  MoveL 676 to (191.54, 223.77, -20.05) mm, rotated rx -180 ry 0 rz 179.9 deg; joints [20.767, -38.825, 103.576, -157.088, 65.575, 170.653]
  MoveL 677 to (191.29, 223.93, -20.05) mm, rotated rx 180 ry 0 rz 179.9 deg; joints [20.765, -38.836, 103.603, -157.094, 65.589, 170.66]
  MoveL 678 to (191.03, 224.08, -20.05) mm, rotated rx 180 ry 0 rz 179.9 deg; joints [20.763, -38.848, 103.63, -157.098, 65.603, 170.667]
  MoveL 679 to (190.78, 224.2, -20.05) mm, rotated rx -180 ry 0 rz 179.9 deg; joints [20.762, -38.859, 103.656, -157.102, 65.617, 170.674]
  MoveL 680 to (190.53, 224.3, -20.05) mm, rotated rx 180 ry 0 rz 179.9 deg; joints [20.762, -38.87, 103.681, -157.105, 65.63, 170.681]
  MoveL 681 to (190.28, 224.39, -20.05) mm, rotated rx -180 ry 0 rz 179.9 deg; joints [20.762, -38.88, 103.706, -157.107, 65.643, 170.686]
  MoveL 682 to (190.02, 224.47, -20.05) mm, rotated rx -180 ry 0 rz 179.9 deg; joints [20.763, -38.891, 103.731, -157.109, 65.656, 170.692]
  MoveL 683 to (189.72, 224.54, -20.05) mm, rotated rx 180 ry 0 rz 179.9 deg; joints [20.765, -38.903, 103.759, -157.11, 65.672, 170.699]
  MoveL 684 to (189.41, 224.59, -20.05) mm, rotated rx -180 ry 0 rz 179.9 deg; joints [20.767, -38.915, 103.788, -157.11, 65.687, 170.704]
  MoveL 685 to (189.1, 224.63, -20.05) mm, rotated rx 180 ry 0 rz 179.9 deg; joints [20.77, -38.927, 103.815, -157.11, 65.702, 170.71]
  MoveL 686 to (188.8, 224.64, -20.05) mm, rotated rx -180 ry 0 rz 179.9 deg; joints [20.774, -38.939, 103.842, -157.108, 65.717, 170.715]
  MoveL 687 to (187.57, 224.64, -20.05) mm, rotated rx 180 ry 0 rz 179.9 deg; joints [20.79, -38.984, 103.949, -157.101, 65.775, 170.734]
  MoveL 688 to (-182.67, 224.64, -20.05) mm, rotated rx -180 ry 0 rz 179.9 deg; joints [27.375, -50.07, 132.248, -152.35, 82.128, 176.591]
  MoveL 689 to (-188.8, 224.64, -20.05) mm, rotated rx 180 ry 0 rz 179.9 deg; joints [27.516, -50.21, 132.665, -152.225, 82.383, 176.704]
  MoveL 690 to (-189.1, 224.63, -20.05) mm, rotated rx -180 ry 0 rz 179.9 deg; joints [27.524, -50.217, 132.685, -152.219, 82.395, 176.71]
  MoveL 691 to (-189.41, 224.59, -20.05) mm, rotated rx -180 ry 0 rz 179.9 deg; joints [27.532, -50.223, 132.705, -152.211, 82.407, 176.715]
  MoveL 692 to (-189.72, 224.54, -20.05) mm, rotated rx 180 ry 0 rz 179.9 deg; joints [27.542, -50.23, 132.724, -152.202, 82.419, 176.72]
  MoveL 693 to (-190.02, 224.47, -20.05) mm, rotated rx 180 ry 0 rz 179.9 deg; joints [27.552, -50.236, 132.742, -152.192, 82.43, 176.724]
  MoveL 694 to (-190.28, 224.39, -20.05) mm, rotated rx -180 ry 0 rz 179.9 deg; joints [27.561, -50.241, 132.757, -152.184, 82.439, 176.728]
  MoveL 695 to (-190.53, 224.3, -20.05) mm, rotated rx -180 ry 0 rz 179.9 deg; joints [27.571, -50.245, 132.771, -152.174, 82.448, 176.731]
  MoveL 696 to (-190.78, 224.2, -20.05) mm, rotated rx -180 ry 0 rz 179.9 deg; joints [27.582, -50.25, 132.784, -152.164, 82.457, 176.734]
  MoveL 697 to (-191.03, 224.08, -20.05) mm, rotated rx -180 ry 0 rz 179.9 deg; joints [27.593, -50.254, 132.797, -152.153, 82.465, 176.736]
  MoveL 698 to (-191.28, 223.93, -20.05) mm, rotated rx 180 ry 0 rz 179.9 deg; joints [27.605, -50.258, 132.809, -152.142, 82.473, 176.739]
  MoveL 699 to (-191.54, 223.77, -20.05) mm, rotated rx -180 ry 0 rz 179.9 deg; joints [27.618, -50.262, 132.82, -152.129, 82.48, 176.741]
  MoveL 700 to (-191.79, 223.59, -20.05) mm, rotated rx 180 ry 0 rz 179.9 deg; joints [27.632, -50.266, 132.831, -152.115, 82.487, 176.743]
  MoveL 701 to (-192.04, 223.38, -20.05) mm, rotated rx 180 ry 0 rz 179.9 deg; joints [27.647, -50.269, 132.841, -152.1, 82.493, 176.744]
  MoveL 702 to (-192.27, 223.16, -20.05) mm, rotated rx -180 ry 0 rz 179.9 deg; joints [27.662, -50.272, 132.849, -152.086, 82.499, 176.744]
  MoveL 703 to (-192.48, 222.94, -20.05) mm, rotated rx -180 ry 0 rz 179.9 deg; joints [27.677, -50.274, 132.855, -152.071, 82.503, 176.745]
  MoveL 704 to (-192.68, 222.69, -20.05) mm, rotated rx -180 ry 0 rz 179.9 deg; joints [27.693, -50.276, 132.86, -152.055, 82.507, 176.744]
  MoveL 705 to (-192.86, 222.44, -20.05) mm, rotated rx 180 ry 0 rz 179.9 deg; joints [27.708, -50.278, 132.863, -152.04, 82.51, 176.743]
  MoveL 706 to (-193.02, 222.19, -20.05) mm, rotated rx -180 ry 0 rz 179.9 deg; joints [27.723, -50.278, 132.865, -152.025, 82.511, 176.742]
  MoveL 707 to (-193.16, 221.93, -20.05) mm, rotated rx -180 ry 0 rz 179.9 deg; joints [27.738, -50.279, 132.865, -152.01, 82.512, 176.741]
  MoveL 708 to (-193.29, 221.68, -20.05) mm, rotated rx -180 ry 0 rz 179.9 deg; joints [27.752, -50.279, 132.865, -151.996, 82.513, 176.739]
  MoveL 709 to (-193.39, 221.43, -20.05) mm, rotated rx -180 ry 0 rz 179.9 deg; joints [27.765, -50.278, 132.863, -151.982, 82.512, 176.736]
  MoveL 710 to (-193.48, 221.18, -20.05) mm, rotated rx 180 ry 0 rz 179.9 deg; joints [27.779, -50.278, 132.86, -151.969, 82.511, 176.734]
  MoveL 711 to (-193.55, 220.92, -20.05) mm, rotated rx 180 ry 0 rz 179.9 deg; joints [27.792, -50.277, 132.856, -151.956, 82.509, 176.731]
  MoveL 712 to (-193.62, 220.62, -20.05) mm, rotated rx 180 ry 0 rz 179.9 deg; joints [27.807, -50.275, 132.85, -151.94, 82.506, 176.727]
  MoveL 713 to (-193.68, 220.31, -20.05) mm, rotated rx -180 ry 0 rz 179.9 deg; joints [27.822, -50.273, 132.842, -151.925, 82.502, 176.723]
  MoveL 714 to (-193.71, 220, -20.05) mm, rotated rx 180 ry 0 rz 179.9 deg; joints [27.836, -50.27, 132.833, -151.91, 82.498, 176.718]
  MoveL 715 to (-193.72, 219.7, -20.05) mm, rotated rx 180 ry 0 rz 179.9 deg; joints [27.85, -50.267, 132.823, -151.896, 82.493, 176.713]
  MoveL 716 to (-193.72, 216.02, -20.05) mm, rotated rx 180 ry 0 rz 179.9 deg; joints [28.013, -50.226, 132.691, -151.726, 82.422, 176.651]
  MoveL 717 to (-193.72, 215.4, -20.05) mm, rotated rx -180 ry 0 rz 179.9 deg; joints [28.04, -50.219, 132.669, -151.698, 82.41, 176.64]
  MoveL 718 to (-193.7, 215.09, -20.05) mm, rotated rx -180 ry 0 rz 179.9 deg; joints [28.053, -50.215, 132.657, -151.684, 82.404, 176.635]
  MoveL 719 to (-193.67, 214.79, -20.05) mm, rotated rx 180 ry 0 rz 179.9 deg; joints [28.066, -50.211, 132.643, -151.671, 82.396, 176.629]
  MoveL 720 to (-192.47, 207.26, -20.05) mm, rotated rx -180 ry 0 rz 179.9 deg; joints [28.368, -50.1, 132.29, -151.35, 82.203, 176.477]
  MoveL 721 to (-126.84, -206.97, -20.05) mm, rotated rx 180 ry 0 rz 179.9 deg; joints [41.693, -41.06, 108.099, -135.687, 72.167, 164.396]
  MoveL 722 to (-126.77, -207.43, -20.05) mm, rotated rx 180 ry 0 rz 179.9 deg; joints [41.705, -41.046, 108.066, -135.671, 72.156, 164.379]
  MoveC 723 to (-127, -208.24, -20.05) mm, rotated rx 180 ry 0 rz 179.9 deg; joints [41.735, -41.033, 108.034, -135.636, 72.151, 164.356] to (-127.77, -208.59, -20.05) mm, rotated rx 180 ry 0 rz 179.9 deg; joints [41.766, -41.047, 108.065, -135.609, 72.172, 164.36]
  MoveL 724 to (-132.34, -208.5, -20.05) mm, rotated rx 180 ry 0 rz 179.9 deg; joints [41.884, -41.179, 108.375, -135.53, 72.331, 164.456]
  MoveC 725 to (-133.05, -208.49, -19.76) mm, rotated rx -180 ry 0 rz 179.9 deg; joints [41.902, -41.216, 108.426, -135.514, 72.346, 164.461] to (-133.34, -208.48, -19.05) mm, rotated rx -180 ry 0 rz 179.9 deg; joints [41.91, -41.265, 108.453, -135.502, 72.332, 164.443]
  Set speed (100.0 mm/s)
  MoveL 726 to (-133.34, -208.48, 15) mm, rotated rx 180 ry 0 rz 179.9 deg; joints [41.891, -43.185, 108.764, -135.148, 71.183, 163.257]
  MoveL 727 to (-133.34, -208.48, 15) mm, rotated rx 180 ry 0 rz 179.9 deg; joints [41.891, -43.185, 108.764, -135.148, 71.183, 163.257]
